TYPE ST_DISDiagnosisMX :
STRUCT
	bWirebreakCh1 AT%I* : BOOL;
	bWirebreakCh2 AT%I* : BOOL;
	bWirebreakCh3 AT%I* : BOOL;
	bWirebreakCh4 AT%I* : BOOL;
	bWirebreakCh5 AT%I* : BOOL;
	bWirebreakCh6 AT%I* : BOOL;
	bWirebreakCh7 AT%I* : BOOL;
	bWirebreakCh8 AT%I* : BOOL;
END_STRUCT
END_TYPE

(* stored: Version 1.1.0.1
   DUT ST_DISDiagnosisMX: Id {43fdaa55-2e59-4bc0-9333-9e4ad9826933} *)
